{attribute 'GeneratedUsingTerminal: EJ7211-0010-0026'}
{attribute addProperty BoxType "EJ7211-0010-0026"}
{attribute addProperty Id "StatuswordAT %I*UINT2"}
{attribute addProperty CRC "2604072444"}
{attribute addProperty Size "2"}
TYPE DRV_Statusword_9B36FDFC EXTENDS InputBase_8311D824 :
STRUCT
	{attribute addProperty Name "Statusword"}
	Statusword AT %I* : UINT;
END_STRUCT
END_TYPE

(* stored: Version 1.2.0.0, ProductVersion 3.1.4024.9
   DUT DRV_Statusword_9B36FDFC: Id {801df7a4-08d4-4be2-b956-d2baa023f7c3} *)
